INTERFACE I_AxisRef

PROPERTY Axis : REFERENCE TO AXIS_REF
GET
END_GET
END_PROPERTY

END_INTERFACE

(* stored: Version 1.1.0.1, ProductVersion 3.1.4026.18
   Itf I_AxisRef: Id {5d39cf7c-0ebc-472e-8bda-dba8743e6161}
   Property Axis: Id {779572b4-cd4b-4727-86ba-7e22b0f7ace6}
   Get Get: Id {694871a5-2f52-4f47-b827-343eb42ef703} *)
